// TIA Portal V20 export
TYPE "LER_typeSequenceInterface"
// stored: Access Published
   STRUCT
      jobs : "LAF_typeJobsInterface";
      sequence : "LAF_typeSequenceInterface";
   END_STRUCT;
END_TYPE
